RoboDK station: assembly.rdk

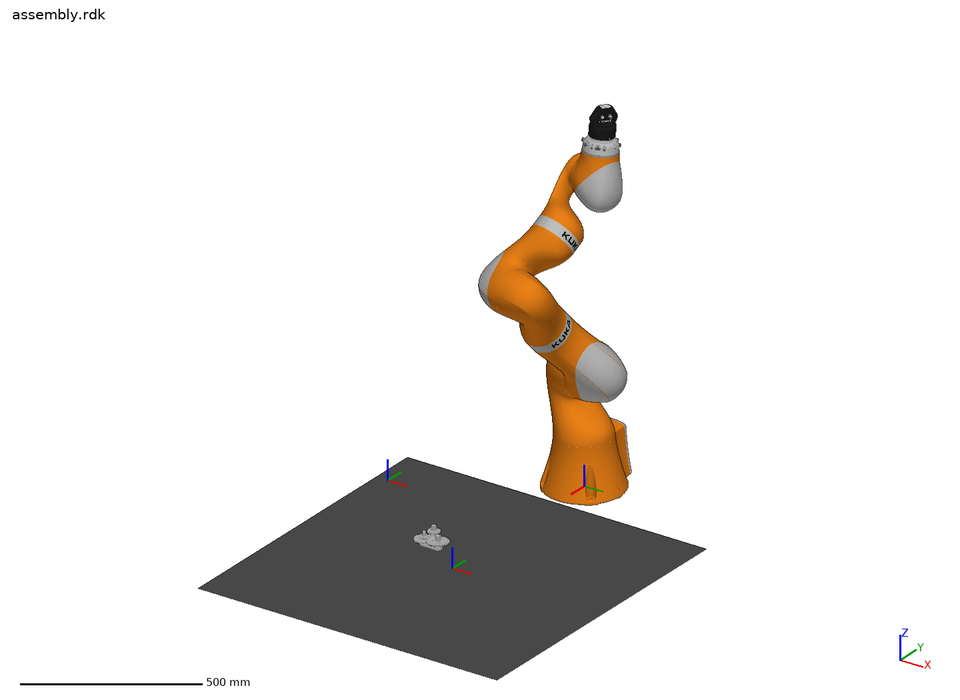
[picture v0: the station drawn from its stored meshes, robots at their saved joint values, targets as dots, program paths as lines]
Station assembly (saved by RoboDK 5.2.1). Poses are relative to the parent item; angles as X-Y-Z fixed-axis rotations.
Station parameters (name, value as stored): AutoAvoidance, YuMi IRB 14000-0.5/0.5-R, AutoAvoidance-Rob YuMi IRB 14000-0.5/0.5-R
  - frame workspace at (0, 0, 200) mm
    - object assembly_place at (0, 0, 0) mm, size 1000 x 1000 x 0.5 mm, geometry from plane_1m.sld
      - object base_plate at (-150, 80, 0) mm, size 71.4 x 71.9 x 41 mm, geometry from base_plate.stl
      - object compound_gear at (-150, 80, 15) mm, size 60.6 x 60.6 x 11.4 mm, geometry from compound_gear.stl
      - object shaft1 at (-150, 126, 41) mm, rotated rx 180 ry 0 rz 180 deg, size 12 x 12 x 38.5 mm, geometry from shaft1.stl
      - object shaft2 at (-104, 80, 41) mm, rotated rx 180 ry 0 rz -180 deg, size 14 x 14 x 38.5 mm, geometry from shaft2.stl
      - object gear1 at (-150, 126, 20) mm, size 39.6 x 39.4 x 5.4 mm, geometry from gear1.stl
      - object gear2 at (-104, 80, 20) mm, size 64.9 x 64.9 x 5.4 mm, geometry from gear2.stl
  - frame KUKA LBR iiwa 14 R820 Base at (0, 630, 200) mm, rotated rx 0 ry 0 rz -90 deg
    - robot robot (model KUKA LBR iiwa 14 R820): 7 axes, payload 14 kg, reach 820 mm, repeatability 0.1 mm, weight 29.9 kg
        modified DH rows (alpha deg, a mm, theta deg, d mm): 0, 0, 0, 360; -90, 0, 0, 0; 90, 0, 0, 420; -90, 0, 0, 0; 90, 0, 0, 400; -90, 0, 0, 0; 90, 0, 0, 126
        joint limits [-170, -120, -170, -120, -170, -120, -175] to [170, 120, 170, 120, 170, 120, 175]; home [0, 0, 0, -90, 0, 0, 0]; saved at [-10.708, 40, 0, -93.578, 0, 46.422, 169.292]
      - robot RobotiQ 2F85: 1 axes, payload 5 kg
          joint limits [0] to [85]; home [85]; saved at [19.65]
      - tool tcp, TCP at (0, 0, 100) mm
  - frame parts_ref at (-460, 350, 200) mm
